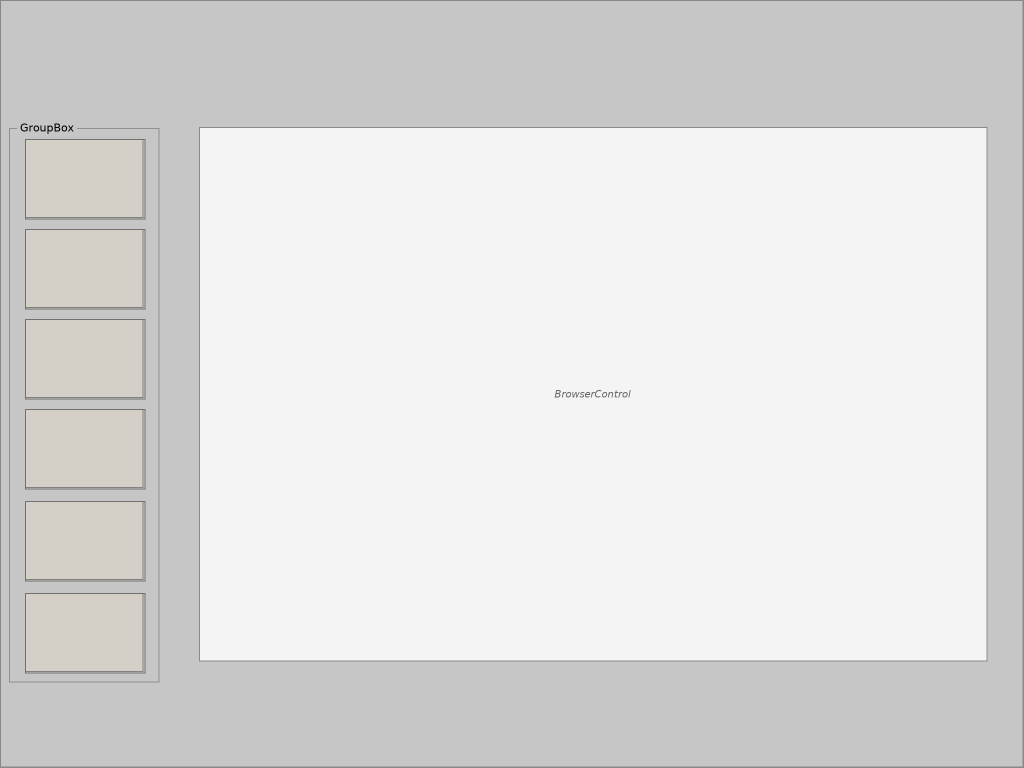
VISUALIZATION Web_300_Browser  // 1024x768
    Frame (0,0 1024x768)
        shows Tmp_000_Template(header := gHMIData.hmiHeader)
    GroupBox (9,120 150x562), "GroupBox"
        Button (16,19 120x80), text list: ''
        Button (16,109 120x80), text list: ''
        Button (16,199 120x80), text list: ''
        Button (16,289 120x80), text list: ''
        Button (16,381 120x80), text list: ''
        Button (16,473 120x80), text list: ''
    BrowserControl (199,127 788x534)
END_VISUALIZATION

(* stored: Version 1.1.0.1, ProductVersion 3.1.4024.11
   Visu Web_300_Browser: Id {314b23d8-2a0f-0237-3a81-4059211f3e27} *)
